// TwinCAT 3 PLC project ServerWritingData
// ProgramVersion: 3.1.4022.2
// libraries:
//   Tc2_Standard, * (Beckhoff Automation GmbH)
//   Tc2_System, * (Beckhoff Automation GmbH)
//   Tc3_Database, * (Beckhoff Automation GmbH)
//   Tc3_IotBase, * (Beckhoff Automation GmbH)
//   Tc3_JsonXml, * (Beckhoff Automation GmbH)
//   Tc3_Module, * (Beckhoff Automation GmbH)
// project tree:
//   DUTs/ ST_Record.TcDUT
//   / PlcTask.TcTTO
//   POUs/ MAIN.TcPOU, PrgMqttCom.TcPOU

CONFIGURATION ServerWritingData
    RESOURCE PLC ON TwinCAT3
        TASK PlcTask(INTERVAL := T#10ms, PRIORITY := 20);
        PROGRAM MAIN WITH PlcTask : MAIN;
    END_RESOURCE
END_CONFIGURATION

// ---- DUTs/ST_Record.TcDUT
TYPE ST_Record :
STRUCT
	dtTimestamp : DATE_AND_TIME;
    //nID        : LINT;
    sMessage      : REAL;
END_STRUCT
END_TYPE

// ---- POUs/MAIN.TcPOU
PROGRAM MAIN
VAR
	x : INT;
END_VAR

x := x + 1;

PrgMqttCom();
//Read_Write_DB();

END_PROGRAM

// ---- POUs/PrgMqttCom.TcPOU
PROGRAM PrgMqttCom
VAR
	fbMqttClient : FB_IotMqttClient;
	bSetParameter : BOOL := TRUE;
	bConnect : BOOL := TRUE;
	
	(* received message *)
	bSubscribed : BOOL;
	sTopicSub : STRING(255) := 'sensor1';
	{attribute 'TcEncoding':='UTF-8'}
	sTopicRcv : STRING(255);
	{attribute 'TcEncoding':='UTF-8'}
	sPayloadRcv : STRING(255);
	fbMessageQueue : FB_IotMqttMessageQueue;
	fbMessage : FB_IotMqttMessage;
	
	hrErrorOccurred : HRESULT; // contains the latest occurred error
	
	fbPLCDBWrite    :  FB_PLCDBWrite(sNetID := '', tTimeout := T#5S);
    myRecord        :  ST_Record;
    ColumnNames     :  ARRAY[0..2] OF STRING(50);
    
	fbJsonDataType	: FB_JsonReadWriteDataType;
	
	nState : INT := 0;
END_VAR

IF bSetParameter THEN
	bSetParameter := FALSE;
	fbMqttClient.sHostName:= 'localhost';
	fbMqttClient.nHostPort:= 1883;
//	fbMqttClient.sClientId:= 'MyTcMqttClient'; 
	fbMqttClient.sTopicPrefix:= ''; 
//	fbMqttClient.nKeepAlive:= 60; 
//	fbMqttClient.sUserName:= ;
//	fbMqttClient.sUserPassword:= ; 
//	fbMqttClient.stWill:= ; 
//	fbMqttClient.stTLS:= ;
	fbMqttClient.ipMessageQueue := fbMessageQueue;
	
	ColumnNames[0] := 'Timestamp';
	//ColumnNames[1] := 'ID';
	ColumnNames[1] := 'Message';
END_IF

fbMqttClient.Execute(bConnect);
IF fbMqttClient.bError THEN
	// add your error logging here
	hrErrorOccurred := fbMqttClient.hrErrorCode;
END_IF


//if there's a message, read it
IF nState = 0 AND fbMessageQueue.nQueuedMessages > 0 THEN
	IF fbMessageQueue.Dequeue(fbMessage:=fbMessage) THEN
		fbMessage.GetTopic(pTopic:=ADR(sTopicRcv), nTopicSize:=SIZEOF(sTopicRcv) );
		fbMessage.GetPayload(pPayload:=ADR(sPayloadRcv), nPayloadSize:=SIZEOF(sPayloadRcv), bSetNullTermination:=FALSE);
		nState := 10;
	END_IF
END_IF


//write received data to structure
IF nState = 10 THEN
	fbJsonDataType.SetSymbolFromJson(sPayloadRcv, 'ST_Record', SIZEOF(myRecord), ADR(myRecord));
	nState := 20;
END_IF


//write received structure to DB
IF nState = 20 THEN
	IF fbPLCDBWrite.WriteStruct(
		hDBID:= 1, 
		sTableName:= 'table4_autoIncrement', 
		pRecord:= ADR(myRecord), 
		cbRecord:= SIZEOF(myRecord), 
		pColumnNames:= ADR(ColumnNames) , 
		cbColumnNames:= SIZEOF(ColumnNames))
	THEN
		IF fbPLCDBWrite.bError THEN
			nState := 245; 
			//ipResultEvt := fbPLCDBWrite.ipTcResultEvent;
		ELSE
			nState := 0;
		END_IF
	END_IF
END_IF


IF fbMqttClient.bConnected THEN
	IF NOT bSubscribed THEN
		bSubscribed := fbMqttClient.Subscribe(sTopic:=sTopicSub, eQoS:=TcIotMqttQos.AtMostOnceDelivery);
		IF fbMqttClient.bError THEN
			// add your error logging here
			hrErrorOccurred := fbMqttClient.hrErrorCode;
		END_IF
	END_IF
END_IF

END_PROGRAM
